/// enumeration of all possible priority
TYPE E_Priority :
(
	/// no priority
	ePriority_none := 0,
	/// info priority
	ePriority_info := 1,
	/// warn priority
	ePriority_warning := 2,
	/// error priority -> Zyklusstop
	ePriority_fault := 3,
	/// error priority with fast stop -> Stopp im aktuellen Schritt 
	ePriority_faultFastStop := 4,
	/// error priority with emergency stop -> Sofortstop aller Objekte
	ePriority_faultEmergency := 5
);
END_TYPE

(* stored: Version 1.1.0.1
   DUT E_Priority: Id {d87000b8-ce05-4d44-bf53-f177ca41ad18} *)
